{attribute addProperty BoxType "EP6601-0002-0018"}
{attribute addProperty Id "InfoDataInfoData_BC63D37F8010"}
{attribute addProperty CRC "424293389"}
{attribute addProperty SizeInBites "80"}
{attribute addProperty SizeInBytes "10"}
TYPE EP6601_194A340D :
STRUCT
	{attribute addProperty Name "InfoData"}
	InfoData : InfoData_BC63D37F;
END_STRUCT
END_TYPE

(* stored: Version 1.2.0.0, ProductVersion 3.1.4024.9
   DUT EP6601_194A340D: Id {8adf6b9a-d50c-49b1-bde4-6eeb14a49aad} *)
